(* IEC 61131-3 sources: IEC.vim/samples, 2 files *)

(* ---- simple.il ---- *)
PROGRAM program0
  LD   x
  MUL  A
  ADD  B
  ST   Y
END_PROGRAM

CONFIGURATION config

  RESOURCE resource1 ON PLC
    TASK task0(INTERVAL := T#20ms,PRIORITY := 0);
    PROGRAM
        instance0 WITH task0 : program0;
    END_PROGRAM
  END_RESOURCE
END_CONFIGURATION

(* ---- simple.st ---- *)
PROGRAM program0
  VAR
    (* Var1 definition *)
    Var1: DINT;
  END_VAR

  {}
END_PROGRAM

CONFIGURATION config

  RESOURCE resource1 ON PLC
    TASK task0(INTERVAL := T#20ms,PRIORITY := 0);
    PROGRAM instance0 WITH task0 : program0;
  END_RESOURCE
END_CONFIGURATION
